PROGRAM P_Demo_FRAC
VAR
    lrUnixTimeSec   : LREAL := 1715433600.5; // 外部送入的 Unix 秒（含小数）；在线写值模拟不同时间戳
    lrFractionalSec : LREAL; // FRAC 输出：带符号的小数部分
    lrIntegerSec    : LREAL; // LTRUNC 输出：朝零截断的整数部分（与 FRAC 互补）
    nNanosecondPart : DINT; // 小数部分 × 1e9 后的纳秒整数
END_VAR

// =============================================================================
// 场景：上位机送来 LREAL 秒数（如 Unix epoch 1715433600.5），需要拆成
//       "整秒"+"纳秒部分"两份：整秒用于 MES 主键，纳秒部分给质量时序对齐。
//
// 价值：FRAC 一行直接给出带符号的小数部分；与 LTRUNC 互补完成整数+小数拆分。
//       省去自己写 x-LTRUNC(x) 的两步代码。
//
// 验证步骤：
//   1. 引用 Tc2_Math
//   2. 在 PLC 项目右键 → Add Existing Item (.TcPOU) → 选本文件 → OK
//   3. 编译、登录、运行
//   4. 在线 monitor 看：
//      - lrUnixTimeSec = 1715433600.5 → lrFractionalSec = 0.5,
//        lrIntegerSec = 1715433600, nNanosecondPart = 500_000_000
//      - 在线改 1715433600.0 → 0.0 / 1715433600 / 0
//      - 改 -1.25 → -0.25 / -1 / -250_000_000 （验证符号保留）
// =============================================================================

// 单行调用：FRAC 取带符号小数部分；LTRUNC 取朝零截断的整数部分
// 两者相加恒等于 lrUnixTimeSec（LREAL 精度内）
lrFractionalSec := FRAC(lrUnixTimeSec);
lrIntegerSec   := LTRUNC(lrUnixTimeSec);

// 小数秒 × 1e9 转纳秒整数；典型 Unix 时间戳 ~1.7e9 远低于 2^53，安全
nNanosecondPart := LREAL_TO_DINT(lrFractionalSec * 1.0E9);

END_PROGRAM

(* stored: Version 1.1.0.1, ProductVersion 3.1.4024.5
   POU P_Demo_FRAC: Id {d5ee93c4-c2c2-5166-afee-8625cc6d5eff}, SpecialFunc None *)
